// LS Electric XG5000 project: unity
// PLC LSPLC

PROGRAM NewProgram (task: 스캔 프로그램)

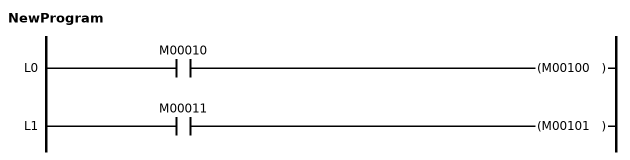
; L0
LOAD      M00010
OUT       M00100
; L1
LOAD      M00011
OUT       M00101